FUNCTION_BLOCK TcoInspectorDialog EXTENDS TcoCore.TcoDialogBase
VAR  
    {attribute clr [CompilerOmits("BuilderPlainer")]}
    _dialogueRetryTask : TcoCore.TcoTask(THIS^);
    {attribute clr [CompilerOmits("BuilderPlainer")]}
    _dialogueTerminateTask : TcoCore.TcoTask(THIS^);
    {attribute clr [CompilerOmits("BuilderPlainer")]}
    _dialogueOverrideTask : TcoCore.TcoTask(THIS^);
    _isOverInspected      : BOOL;
    {attribute 'hide'}
    _refInspector : REFERENCE TO TcoInspector;
END_VAR

SUPER^();

METHOD SetInspector
VAR_INPUT 
	refInspector : REFERENCE TO TcoInspector;
END_VAR
_refInspector REF= refInspector;
END_METHOD

METHOD Show
VAR_INPUT
	inRetryStep : INT;
END_VAR
_isOverInspected := _refInspector.OverInspected;

 IF(_refInspector.Done) THEN		
	IF(_refInspector.Result = eInspectorResult.Failed) THEN
		THIS^.Invoke();
		SUPER^();	
		
		IF(_dialogueRetryTask.Execute()) THEN
			_dialogueRetryTask.DoneWhen(_refInspector.Retry(inRetryStep));
		END_IF
		
		IF(_dialogueTerminateTask.Execute()) THEN
			_dialogueTerminateTask.DoneWhen(_refInspector.Terminate());
		END_IF
		
		IF(_dialogueOverrideTask.Execute()) THEN
			_dialogueOverrideTask.DoneWhen(_refInspector.CarryOn());
		END_IF
	ELSE
		IF(_refInspector.Coordinator <> 0) THEN
			_refInspector.Coordinator.MoveNext();
		END_IF;	
	END_IF;	
END_IF;
END_METHOD

END_FUNCTION_BLOCK

(* stored: Version 1.1.0.1, ProductVersion 3.1.4024.9
   POU TcoInspectorDialog: Id {c6c9fa75-2ded-0851-0bf8-095f61987545}, SpecialFunc None
   Method SetInspector: Id {59f6bb8e-40b5-01f0-1137-0e38be5ca644}
   Method Show: Id {409527dd-7ec4-05bd-0a53-372d7df86c62} *)
